// TIA Portal V18 export
// export: Created 2026-03-12T16:04:35.1863989Z, ExportSetting WithDefaults, DisplayName Totally Integrated Automation Portal, DisplayVersion V18 Update 5, DisplayName TIA Portal Openness, DisplayVersion V18 Update 5, DisplayName TIA Portal Version Control Interface, DisplayVersion V18, DisplayName SINAMICS Startdrive Advanced, DisplayVersion V18, DisplayName SINAMICS Startdrive G130, G150, S120, S150, SINAMICS MV, S210, DisplayVersion V18, DisplayName SINAMICS Startdrive G110M, G120, G120C, G120D, G120P, G115D, DisplayVersion V18, DisplayName STEP 7 Professional, DisplayVersion V18 Update 5, DisplayName STEP 7 Safety, DisplayVersion V18, DisplayName WinCC Professional, DisplayVersion V18 Update 5
FUNCTION_BLOCK "FB FILTRO DE AMOSTRAGEM  ANALÍTICA"   // FB24, LAD
{ S7_Optimized_Access := 'TRUE' }
VERSION : 0.1
// stored: AutoNumber true, IsIECCheckEnabled false, IsRetainMemResEnabled false, MemoryReserve 100, SetENOAutomatically false, UDAEnableTagReadback false
   VAR_INPUT
      INPUT_SENSOR : Int;
   END_VAR
   VAR_OUTPUT
      OUTPUT_SENSOR : Int;
   END_VAR
   VAR
      INDEX_AMOSTRAGEM : Int;
      AUX_1 : Int;
      AUX_2 : Int;
      AUX_3 : Int;
      AUX_4 : Int;
      AUX_5 : Int;
      AUX_6 : Int;
      AUX_7 : Int;
      AUX_8 : Int;
      AUX_9 : Int;
      AUX_10 : Bool;
      AUX_11 : Int;
   END_VAR
   VAR_TEMP   // added for the SCL form of the ladder/FBD networks
      _w1 : Bool;
   END_VAR
BEGIN

REGION Network 1: Sistema de Amostragem
   // O sistema irá realizar 4 amostra no periodo de 2s e realizar um filtro, contra interferências externas no sistema.
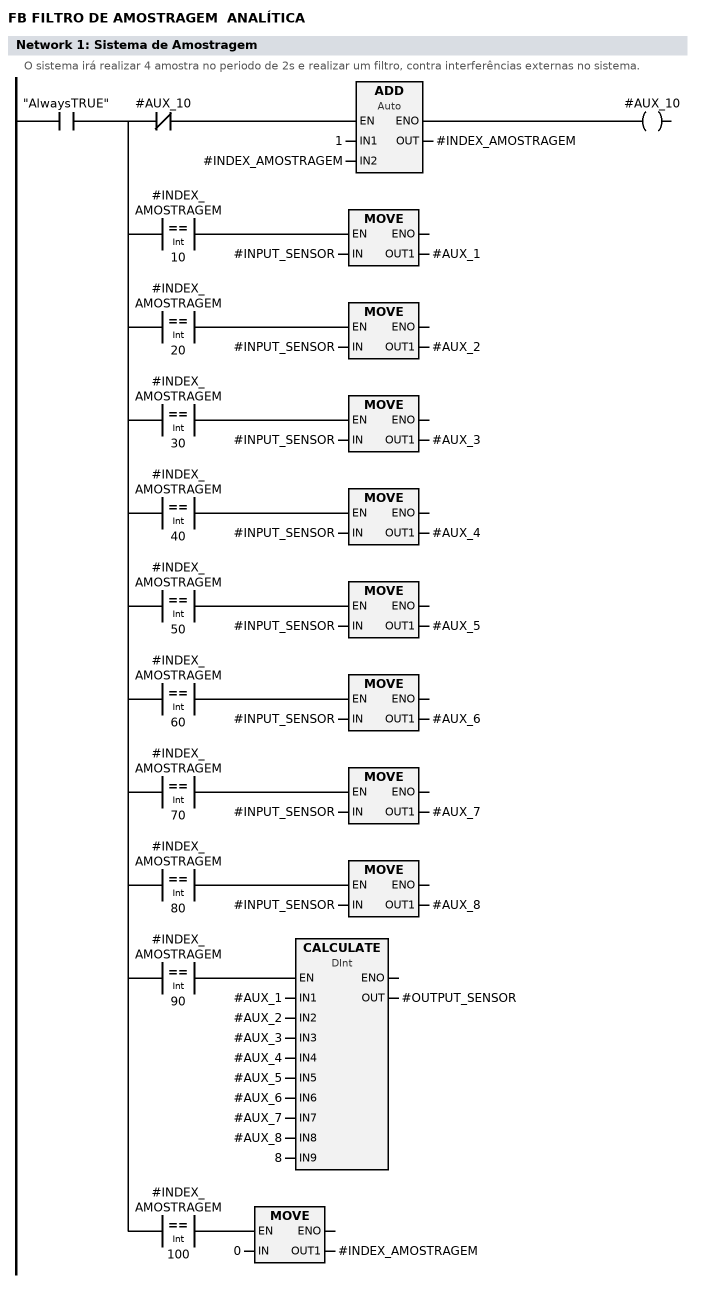
   RUNG wire#powerrail
      Contact( "AlwaysTRUE" )
      wire#w1
      I_Contact( #AUX_10 )
      Add(in1 := 1, in2 := #INDEX_AMOSTRAGEM, out => #INDEX_AMOSTRAGEM)
      Coil( #AUX_10 )
   END_RUNG
   RUNG wire#w1
      { S7_Templates := "SrcType := Int" } EQ_Contact(in1 := #INDEX_AMOSTRAGEM, in2 := 10)
      Move(in := #INPUT_SENSOR, out1 => #AUX_1)
   END_RUNG
   RUNG wire#w1
      { S7_Templates := "SrcType := Int" } EQ_Contact(in1 := #INDEX_AMOSTRAGEM, in2 := 20)
      Move(in := #INPUT_SENSOR, out1 => #AUX_2)
   END_RUNG
   RUNG wire#w1
      { S7_Templates := "SrcType := Int" } EQ_Contact(in1 := #INDEX_AMOSTRAGEM, in2 := 30)
      Move(in := #INPUT_SENSOR, out1 => #AUX_3)
   END_RUNG
   RUNG wire#w1
      { S7_Templates := "SrcType := Int" } EQ_Contact(in1 := #INDEX_AMOSTRAGEM, in2 := 40)
      Move(in := #INPUT_SENSOR, out1 => #AUX_4)
   END_RUNG
   RUNG wire#w1
      { S7_Templates := "SrcType := Int" } EQ_Contact(in1 := #INDEX_AMOSTRAGEM, in2 := 50)
      Move(in := #INPUT_SENSOR, out1 => #AUX_5)
   END_RUNG
   RUNG wire#w1
      { S7_Templates := "SrcType := Int" } EQ_Contact(in1 := #INDEX_AMOSTRAGEM, in2 := 60)
      Move(in := #INPUT_SENSOR, out1 => #AUX_6)
   END_RUNG
   RUNG wire#w1
      { S7_Templates := "SrcType := Int" } EQ_Contact(in1 := #INDEX_AMOSTRAGEM, in2 := 70)
      Move(in := #INPUT_SENSOR, out1 => #AUX_7)
   END_RUNG
   RUNG wire#w1
      { S7_Templates := "SrcType := Int" } EQ_Contact(in1 := #INDEX_AMOSTRAGEM, in2 := 80)
      Move(in := #INPUT_SENSOR, out1 => #AUX_8)
   END_RUNG
   RUNG wire#w1
      { S7_Templates := "SrcType := Int" } EQ_Contact(in1 := #INDEX_AMOSTRAGEM, in2 := 90)
      { S7_Templates := "SrcType := DInt"; S7_Expression := "(IN1+IN2+IN3+IN4+IN5+IN6+IN7+IN8)/IN9" } Calculate(in1 := #AUX_1, in2 := #AUX_2, in3 := #AUX_3, in4 := #AUX_4, in5 := #AUX_5, in6 := #AUX_6, in7 := #AUX_7, in8 := #AUX_8, in9 := 8, out => #OUTPUT_SENSOR)
   END_RUNG
   RUNG wire#w1
      { S7_Templates := "SrcType := Int" } EQ_Contact(in1 := #INDEX_AMOSTRAGEM, in2 := 100)
      Move(in := 0, out1 => #INDEX_AMOSTRAGEM)
   END_RUNG
   // the same network as SCL:
   #_w1 := "AlwaysTRUE" AND NOT #AUX_10;
   IF #_w1 THEN #INDEX_AMOSTRAGEM := 1 + #INDEX_AMOSTRAGEM; END_IF;
   #AUX_10 := #_w1;
   IF "AlwaysTRUE" AND (#INDEX_AMOSTRAGEM = 10) THEN #AUX_1 := #INPUT_SENSOR; END_IF;
   IF "AlwaysTRUE" AND (#INDEX_AMOSTRAGEM = 20) THEN #AUX_2 := #INPUT_SENSOR; END_IF;
   IF "AlwaysTRUE" AND (#INDEX_AMOSTRAGEM = 30) THEN #AUX_3 := #INPUT_SENSOR; END_IF;
   IF "AlwaysTRUE" AND (#INDEX_AMOSTRAGEM = 40) THEN #AUX_4 := #INPUT_SENSOR; END_IF;
   IF "AlwaysTRUE" AND (#INDEX_AMOSTRAGEM = 50) THEN #AUX_5 := #INPUT_SENSOR; END_IF;
   IF "AlwaysTRUE" AND (#INDEX_AMOSTRAGEM = 60) THEN #AUX_6 := #INPUT_SENSOR; END_IF;
   IF "AlwaysTRUE" AND (#INDEX_AMOSTRAGEM = 70) THEN #AUX_7 := #INPUT_SENSOR; END_IF;
   IF "AlwaysTRUE" AND (#INDEX_AMOSTRAGEM = 80) THEN #AUX_8 := #INPUT_SENSOR; END_IF;
   IF "AlwaysTRUE" AND (#INDEX_AMOSTRAGEM = 90) THEN
       #OUTPUT_SENSOR := (#AUX_1+#AUX_2+#AUX_3+#AUX_4+#AUX_5+#AUX_6+#AUX_7+#AUX_8)/8;
   END_IF;
   IF "AlwaysTRUE" AND (#INDEX_AMOSTRAGEM = 100) THEN #INDEX_AMOSTRAGEM := 0; END_IF;
END_REGION
END_FUNCTION_BLOCK
